FUNCTION FN_IntraloxToLane : cLaneSel
VAR_INPUT
	IntraloxLane: DINT;
	LaneConfig: Cmp3LaneSwitchMainConfig;
END_VAR

IF LaneConfig.OutGreenLine = IntraloxLane THEN
	FN_IntraloxToLane := cLaneSel.Green;
ELSIF LaneConfig.OutRedLine = IntraloxLane THEN
	FN_IntraloxToLane := cLaneSel.Red;
ELSIF LaneConfig.OutBlueLine = IntraloxLane THEN
	FN_IntraloxToLane := cLaneSel.Blue;
END_IF

END_FUNCTION

(* stored: Version 1.1.0.1, ProductVersion 3.1.4024.6
   POU FN_IntraloxToLane: Id {b469f63d-dd6a-4d64-9b14-b6c03b2b6947}, SpecialFunc None *)
